(* IEC 61131-3 sources: s7GBRL/src/config, 2 files *)

(* ---- Configuration.st ---- *)
CONFIGURATION PLC_1

    var_global
        //--------------------------------
        // Global variable for Timers
        //--------------------------------

        //--------------------------------------------------
        // programm SPS 2019 Demonstration
        //--------------------------------------------------
        isInitialized : bool;
        GlobalCounter : INT;
    end_var

    task Main(Priority := 1);
    task System(Interval := T#10ms, Priority := 1);

    program Cyclic with Main : ProgGBRL;

END_CONFIGURATION

(* ---- MainLightStack.st ---- *)
PROGRAM ProgGBRL /* name of the program */

    VAR_EXTERNAL
        GlobalCounter : INT;
    END_VAR
    ;

END_PROGRAM
